// SIMATIC S7-200 project (STEP 7-Micro/WIN), CPU 224XP CN REL 02.01

SYMBOL_TABLE USR1
CRC_value        VW2070   // CRC的计算值
CRC_value_out    VW2090   // 调用CRC计算子程序得出的CRC值
TIMES_SENT       VB2001   // 发送记数寄存器
BYTES_REC        VB2002   // 接收的字节数
DATA_SENT        VB2010   // 发送区的起始字节
ADDRESS          VB2031   // 仪表地址
PORT_NUM         VB2005   // 选择的通信端口（PORT0 或PORT1）
END_SYMBOL_TABLE

SYMBOL_TABLE DI
紧急停止             I0.0
电源故障             I0.1
远程启动             I0.2
远程停止             I0.3
END_SYMBOL_TABLE

SYMBOL_TABLE USS 协议
USS_LOW_V        VD1000   // (DWORD)在此键入 USS协议符号的起始地址。
USS_HIGH_V       VD1004
USS_TIME_OUT     VW1008
USS_I_LINE       VW1010
USS_DAT_PTR0     VD1012
USS_ACT_DRV0     VD1016
USS_CUR_DRV0     VD1020
USS_P0           V1024.0
USS_REQ_SNT0     V1024.1
USS_RETRY_P0     VB1025
USS_ERR_CODE     VB1026
USS_CS_D0        VD1027
USS_CS_W0        VW1027
USS_CS_W2        VW1029
USS_CS_B0        VB1027
USS_CS_B1        VB1028
USS_POLL_BUF     VB1031
USS_XMT_0        VB1046
USS_XMT_ADR0     VB1049
USS_X_STWD       VD1056
USS_X_BCC        VB1060
USS_X_DW1        VD1047
USS_X_DW5        VD1051
USS_X_DW9        VD1055
USS_X_DB13       VB1059
USS_RCV_BUF0     VB1061
USS_R_STX        VB1062
USS_R_LGE        VB1063
USS_R_ADR        VB1064
USS_R_STWD       VD1071
USS_R_DW1        VD1062
USS_R_DW5        VD1066
USS_R_DW9        VD1070
USS_R_W13        VW1074
USS_STAT_TAB     VB1076
USS_ADR_P0       VB1396
END_SYMBOL_TABLE

SYMBOL_TABLE DO
启动排架             Q0.0
启动空调             Q0.1
启动空压机            Q0.2
DF1Q             Q0.3
DF2Q             Q0.4
DF3Q             Q0.5
DF4Q             Q0.6
DF5Q             Q0.7
运行Q              Q1.0
报警Q              Q1.1
END_SYMBOL_TABLE

SYMBOL_TABLE  内部
清洗间隔时间           VW4      // 0-999.9s
自动清洗延迟时间         VW6      // 0-1440min
清洗次数             VW8
报警温度设置值          VW12
报警光强度设置值         VW14
报警液位设置值          VW16
电流高报警设定值         VW18
电压高报警设定值         VW20
电压低报警设定值         VW22
温度高停止运行设置值       VW26
温度降允许运行设置值       VW28
光强低_自动清洗设置值      VW30
液位低停止运行设置值       VW34
液位升允许运行设置值       VW36
状态字1_1           VW38
状态字1_2           VW40
状态字2_1           VW42
状态字2_2           VW44
状态字3_1           VW46
状态字3_2           VW48
状态字4_1           VW50
状态字4_2           VW52
其它报警字1           VW54
其它报警字2           VW56
其它报警字3           VW58
累计运行时间（秒）        VW66     // 0-60
累计运行时间（分）        VW68     // 0-60
累计运行时间（时）        VW70     // 0-32767
累计启动次数           VW72     // 0-32767
温度1实时值           VW74
温度2实时值           VW76
光强实时值            VW78
液位实时值            VW80
电压实时值            VW82
电流实时值            VW84
清洗用临时积存1         VW140
清洗用临时积存2         VW142
清洗用临时积存3已清洗次     VW144
模块1通信监测临时        VB150
模块2通信监测临时        VB151
模块3通信监测临时        VB152
模块4通信监测临时        VB153
模块5通信监测临时        VB154
模块6通信监测临时        VB155
温度控制允许           M2.0     // 0为禁止,1为允许
光强度控制允许          M2.1     // 0为禁止,1为允许
液位控制允许           M2.2     // 0为禁止,1为允许
系统控制模式           M2.3     // 0为本地,1为远程
清洗控制模式           M2.4     // 0为手动,1为自动
温度1异常高           M6.0
温度2异常高           M6.1
光强异常低            M6.2
液位异常低            M6.3
未设定清洗参数          M6.4
未设定灯管开参数         M6.5
未设定报警参数          M6.6
允许清洗             M7.0
允许启动灯管           M7.1
中断清洗运行           M7.2
中断灯管运行           M7.3
模块1通信故障          M8.0
模块2通信故障          M8.1
模块3通信故障          M8.2
模块4通信故障          M8.3
模块5通信故障          M8.4
模块6通信故障          M8.5
排架1镇流器故障         M8.6
排架2镇流器故障         M8.7
排架3镇流器故障         M9.0
排架4镇流器故障         M9.1
排架5镇流器故障         M9.2
排架6镇流器故障         M9.3
排架7镇流器故障         M9.4
排架8镇流器故障         M9.5
排架9镇流器故障         M9.6
排架10镇流器故障        M9.7
灯管启动中            M10.0
清洗中              M10.1
空调运行中            M10.2
空压机运行中           M10.3
灯管本地启动           M10.4
灯管本地停止           M10.5
灯管远程启动           M10.6
灯管远程停止           M10.7
开始清洗             M11.1
停止清洗             M11.2
空调启动             M11.3
空调停止             M11.4
报警复位             M11.5
总报警位             M12.0
温度1高报警           M12.1
温度2高报警           M12.2
光强低报警            M12.3
液位低报警            M12.4
I高报警             M12.5
U高报警             M12.6
U低报警             M12.7
电源故障报警           M13.0
温度1输入故障          M13.1
温度2输入故障          M13.2
光强输入故障           M13.3
液位输入故障           M13.4
I输入故障            M13.5
U输入故障            M13.6
状态字1_1映象         MW14
状态字1_2映象         MW16
状态字2_1映象         MW18
状态字2_2映象         MW20
状态字3_1映象         MW22
状态字3_2映象         MW24
状态字4_1映象         MW26
状态字4_2映象         MW28
END_SYMBOL_TABLE

SYMBOL_TABLE AI
温度1AIW           AIW0     // 4------20ma
光强AIW            AIW2     // 0------5v
温度2AIW           AIW4     // 4------20ma
水位AIW            AIW6     // 4------20ma
电压AIW            AIW8     // 4------20ma
电流AIW            AIW10    // 4------20ma
END_SYMBOL_TABLE

ORGANIZATION_BLOCK MAIN:OB1
TITLE= 西门子PLC   RS485通信控制程序 
// 2007-4-25      Ver1.0      by huangyz0810@163.com
// 2007-4-26      Ver1.1      by huangyz0810@163.com
// 2007-4-30      Ver1.2      by huangyz0810@163.com
// 2007-5-07      Ver1.3      by huangyz0810@163.com
// *************************************************************************************************************************************************
// 注：主程序包括以下程序调用：通信初始化（INIT）、仪表数据处理（DI_DATA）、控制程序（CONTROL）
//         一般设备的控制程序请写入到CONTROL子程序里面。
// 
//         VB2060----VB2099范围内的40个字节空间已经分配给CRC校验子程序,切勿在其它程序中占用,否则引起麻烦
// 
//         VB2000----VB2049范围内的60个字节空间已经分配给通信中断,指针,字节计数等程序,切勿在其它程序中占用,
//                        其中,VB2010----2029 为发送缓冲区
//                                 VB2030----2059 为接收缓冲区
// 
//          VB2100----VB2199范围内的100个字节空间已经分配给数据读取队列,切勿在其它程序中占用,
//                        其中,VB2100----2109 为第数据队列的中间缓冲区
//                                 VB2110----2119 为第一个数据队列
//                                 VB2120----2129 为第二个数据队列
//                                  其它类推。该范围内最多支持9个队列，即最多支持不超过9次通信的设备数量。
//                                 如果需要超过9次通信，需要在 VB2200或其它未使用区域再分配通信队列寄存区
// *************************************************************************************************************************************************
// 
BEGIN
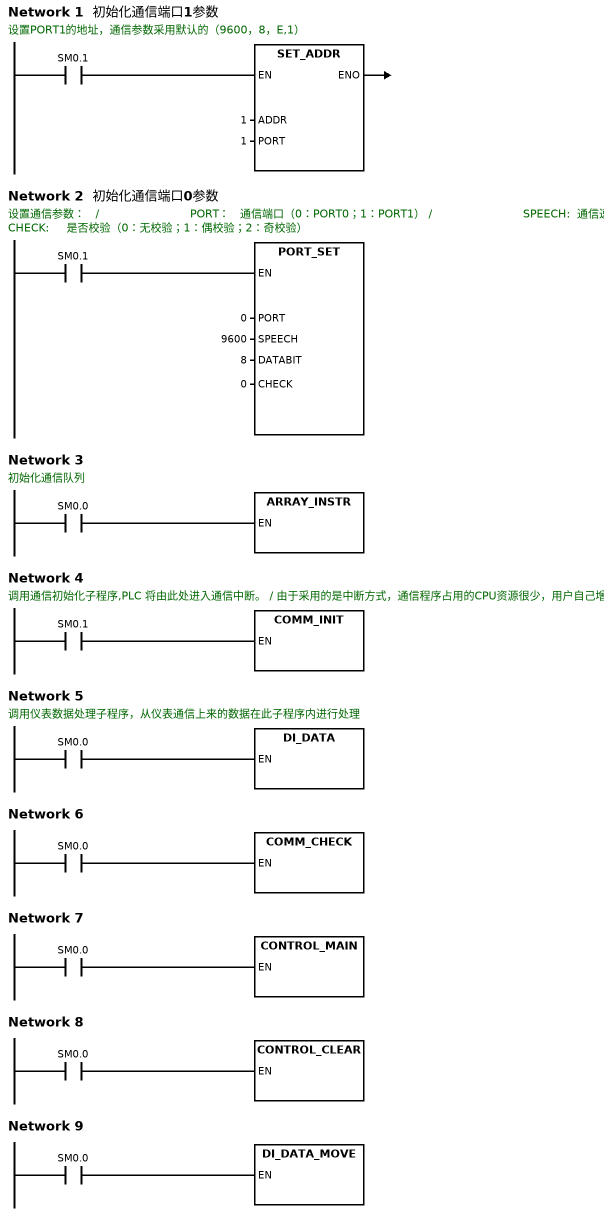
Network 1 // 初始化通信端口1参数
// 设置PORT1的地址，通信参数采用默认的（9600，8，E,1）
LD     SM0.1
SPA    1, 1
Network 2 // 初始化通信端口0参数
// 设置通信参数：  
//                          PORT：   通信端口（0：PORT0；1：PORT1）
//                          SPEECH:  通信速率（1200，2400，4800，9600，19200）
//                          DATABIT  :数据位（7或8）
//                          CHECK:     是否校验（0：无校验；1：偶校验；2：奇校验）
LD     SM0.1
CALL   PORT_SET:SBR55, 0, 9600, 8, 0
Network 3
// 初始化通信队列
LD     SM0.0
CALL   ARRAY_INSTR:SBR60
Network 4
// 调用通信初始化子程序,PLC 将由此处进入通信中断。
// 由于采用的是中断方式，通信程序占用的CPU资源很少，用户自己增加的程序可以很好的使用CPU资源
LD     SM0.1
CALL   COMM_INIT:SBR50
Network 5
// 调用仪表数据处理子程序，从仪表通信上来的数据在此子程序内进行处理
LD     SM0.0
CALL   DI_DATA:SBR52
Network 6
LD     SM0.0
CALL   COMM_CHECK:SBR53
Network 7
LD     SM0.0
CALL   CONTROL_MAIN:SBR1
Network 8
LD     SM0.0
CALL   CONTROL_CLEAR:SBR2
Network 9
LD     SM0.0
CALL   DI_DATA_MOVE:SBR6
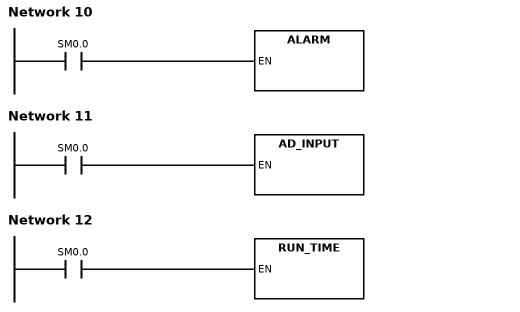
Network 10
LD     SM0.0
CALL   ALARM:SBR7
Network 11
LD     SM0.0
CALL   AD_INPUT:SBR8
Network 12
LD     SM0.0
CALL   RUN_TIME:SBR5
END_ORGANIZATION_BLOCK

SUBROUTINE_BLOCK CONTROL_MAIN:SBR1
TITLE=
BEGIN
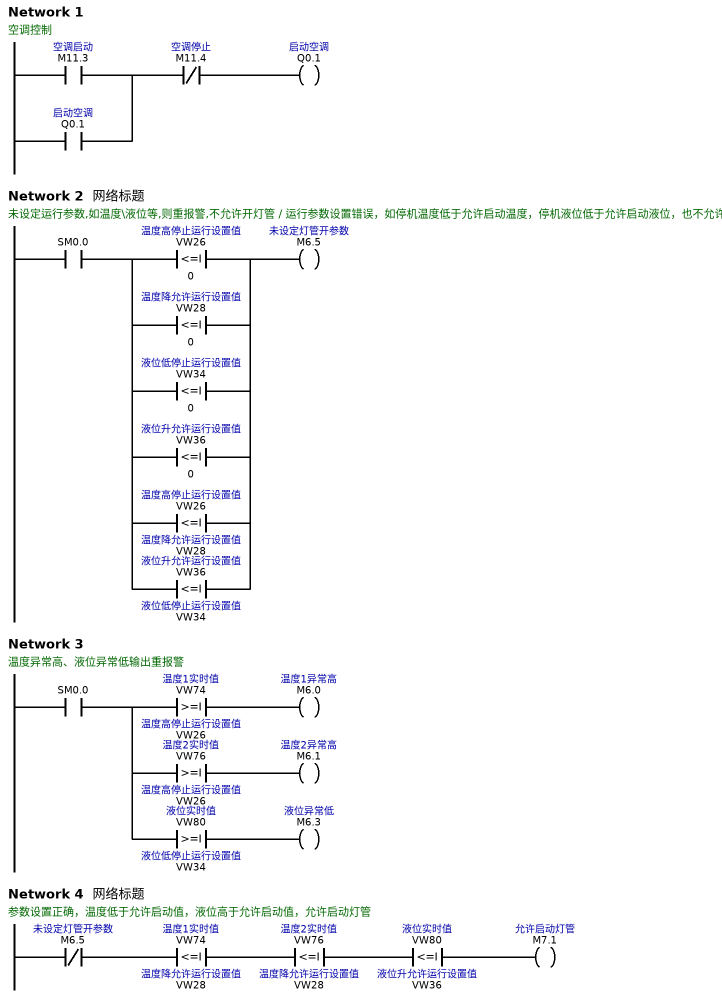
Network 1
// 空调控制
LD     空调启动:M11.3
O      启动空调:Q0.1
AN     空调停止:M11.4
=      启动空调:Q0.1
Network 2 // 网络标题
// 未设定运行参数,如温度\液位等,则重报警,不允许开灯管
// 运行参数设置错误，如停机温度低于允许启动温度，停机液位低于允许启动液位，也不允许开灯管
LD     SM0.0
LDW<=  温度高停止运行设置值:VW26, 0
OW<=   温度降允许运行设置值:VW28, 0
OW<=   液位低停止运行设置值:VW34, 0
OW<=   液位升允许运行设置值:VW36, 0
OW<=   温度高停止运行设置值:VW26, 温度降允许运行设置值:VW28
OW<=   液位升允许运行设置值:VW36, 液位低停止运行设置值:VW34
ALD
=      未设定灯管开参数:M6.5
Network 3
// 温度异常高、液位异常低输出重报警
LD     SM0.0
LPS
AW>=   温度1实时值:VW74, 温度高停止运行设置值:VW26
=      温度1异常高:M6.0
LRD
AW>=   温度2实时值:VW76, 温度高停止运行设置值:VW26
=      温度2异常高:M6.1
LPP
AW>=   液位实时值:VW80, 液位低停止运行设置值:VW34
=      液位异常低:M6.3
Network 4 // 网络标题
// 参数设置正确，温度低于允许启动值，液位高于允许启动值，允许启动灯管
LDN    未设定灯管开参数:M6.5
AW<=   温度1实时值:VW74, 温度降允许运行设置值:VW28
AW<=   温度2实时值:VW76, 温度降允许运行设置值:VW28
AW<=   液位实时值:VW80, 液位升允许运行设置值:VW36
=      允许启动灯管:M7.1
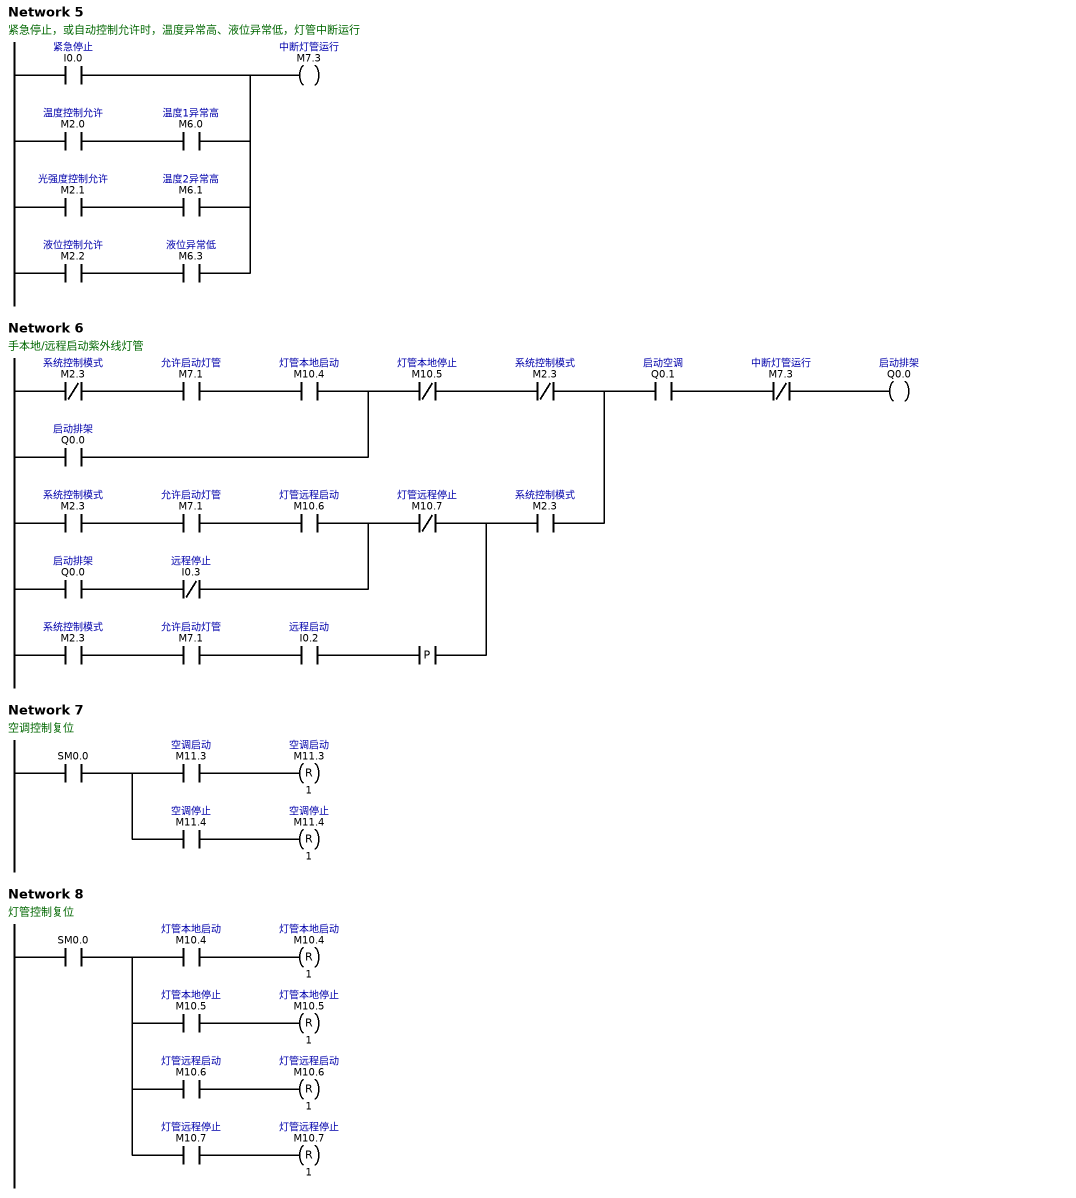
Network 5
// 紧急停止，或自动控制允许时，温度异常高、液位异常低，灯管中断运行
LD     紧急停止:I0.0
LD     温度控制允许:M2.0
A      温度1异常高:M6.0
OLD
LD     光强度控制允许:M2.1
A      温度2异常高:M6.1
OLD
LD     液位控制允许:M2.2
A      液位异常低:M6.3
OLD
=      中断灯管运行:M7.3
Network 6
// 手本地/远程启动紫外线灯管
LDN    系统控制模式:M2.3
A      允许启动灯管:M7.1
A      灯管本地启动:M10.4
O      启动排架:Q0.0
AN     灯管本地停止:M10.5
AN     系统控制模式:M2.3
LD     系统控制模式:M2.3
A      允许启动灯管:M7.1
A      灯管远程启动:M10.6
LD     启动排架:Q0.0
AN     远程停止:I0.3
OLD
AN     灯管远程停止:M10.7
LD     系统控制模式:M2.3
A      允许启动灯管:M7.1
A      远程启动:I0.2
EU
OLD
A      系统控制模式:M2.3
OLD
A      启动空调:Q0.1
AN     中断灯管运行:M7.3
=      启动排架:Q0.0
Network 7
// 空调控制复位
LD     SM0.0
LPS
A      空调启动:M11.3
R      空调启动:M11.3, 1
LPP
A      空调停止:M11.4
R      空调停止:M11.4, 1
Network 8
// 灯管控制复位
LD     SM0.0
LPS
A      灯管本地启动:M10.4
R      灯管本地启动:M10.4, 1
LRD
A      灯管本地停止:M10.5
R      灯管本地停止:M10.5, 1
LRD
A      灯管远程启动:M10.6
R      灯管远程启动:M10.6, 1
LPP
A      灯管远程停止:M10.7
R      灯管远程停止:M10.7, 1
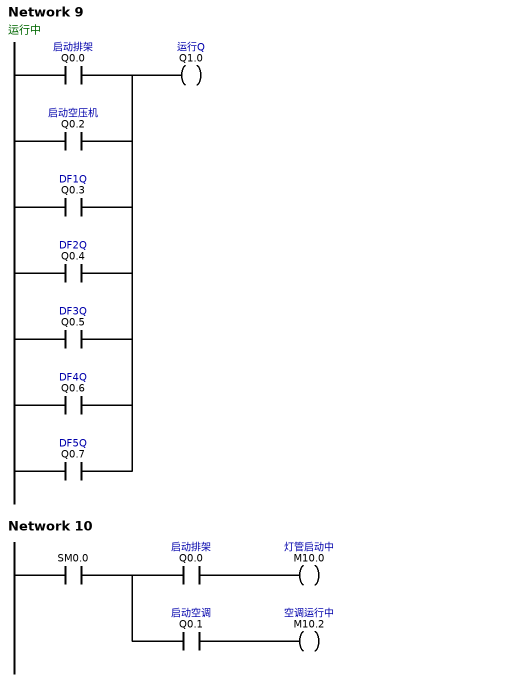
Network 9
// 运行中
LD     启动排架:Q0.0
O      启动空压机:Q0.2
O      DF1Q:Q0.3
O      DF2Q:Q0.4
O      DF3Q:Q0.5
O      DF4Q:Q0.6
O      DF5Q:Q0.7
=      运行Q:Q1.0
Network 10
LD     SM0.0
LPS
A      启动排架:Q0.0
=      灯管启动中:M10.0
LPP
A      启动空调:Q0.1
=      空调运行中:M10.2
END_SUBROUTINE_BLOCK

SUBROUTINE_BLOCK CONTROL_CLEAR:SBR2
TITLE=手动清洗, 清洗模式为"手动"后,先开空压机,延时5分钟,DF1输出10秒（值可调），停止10秒（值可调），反复3次，然后DF2输出10秒（值可调），停止10秒（值可调），反复3次，DF3、DF4、DF5照次类推
VAR
clean_time:WORD;	// LW0 
END_VAR
BEGIN
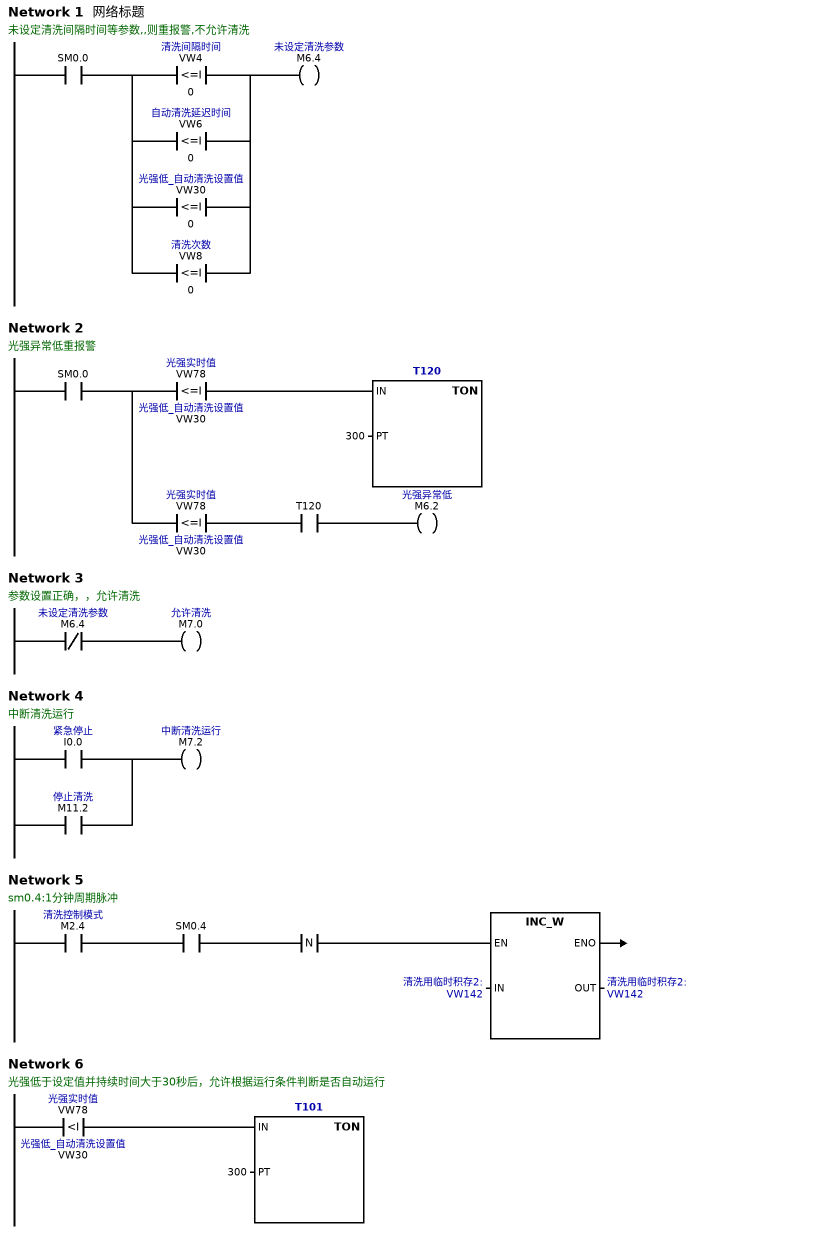
Network 1 // 网络标题
// 未设定清洗间隔时间等参数,,则重报警,不允许清洗
LD     SM0.0
LDW<=  清洗间隔时间:VW4, 0
OW<=   自动清洗延迟时间:VW6, 0
OW<=   光强低_自动清洗设置值:VW30, 0
OW<=   清洗次数:VW8, 0
ALD
=      未设定清洗参数:M6.4
Network 2
// 光强异常低重报警
LD     SM0.0
LPS
AW<=   光强实时值:VW78, 光强低_自动清洗设置值:VW30
TON    T120, 300
LPP
AW<=   光强实时值:VW78, 光强低_自动清洗设置值:VW30
A      T120
=      光强异常低:M6.2
Network 3
// 参数设置正确，，允许清洗
LDN    未设定清洗参数:M6.4
=      允许清洗:M7.0
Network 4
// 中断清洗运行
LD     紧急停止:I0.0
O      停止清洗:M11.2
=      中断清洗运行:M7.2
Network 5
// sm0.4:1分钟周期脉冲
LD     清洗控制模式:M2.4
A      SM0.4
ED
INCW   清洗用临时积存2:VW142
Network 6
// 光强低于设定值并持续时间大于30秒后，允许根据运行条件判断是否自动运行
LDW<   光强实时值:VW78, 光强低_自动清洗设置值:VW30
TON    T101, 300
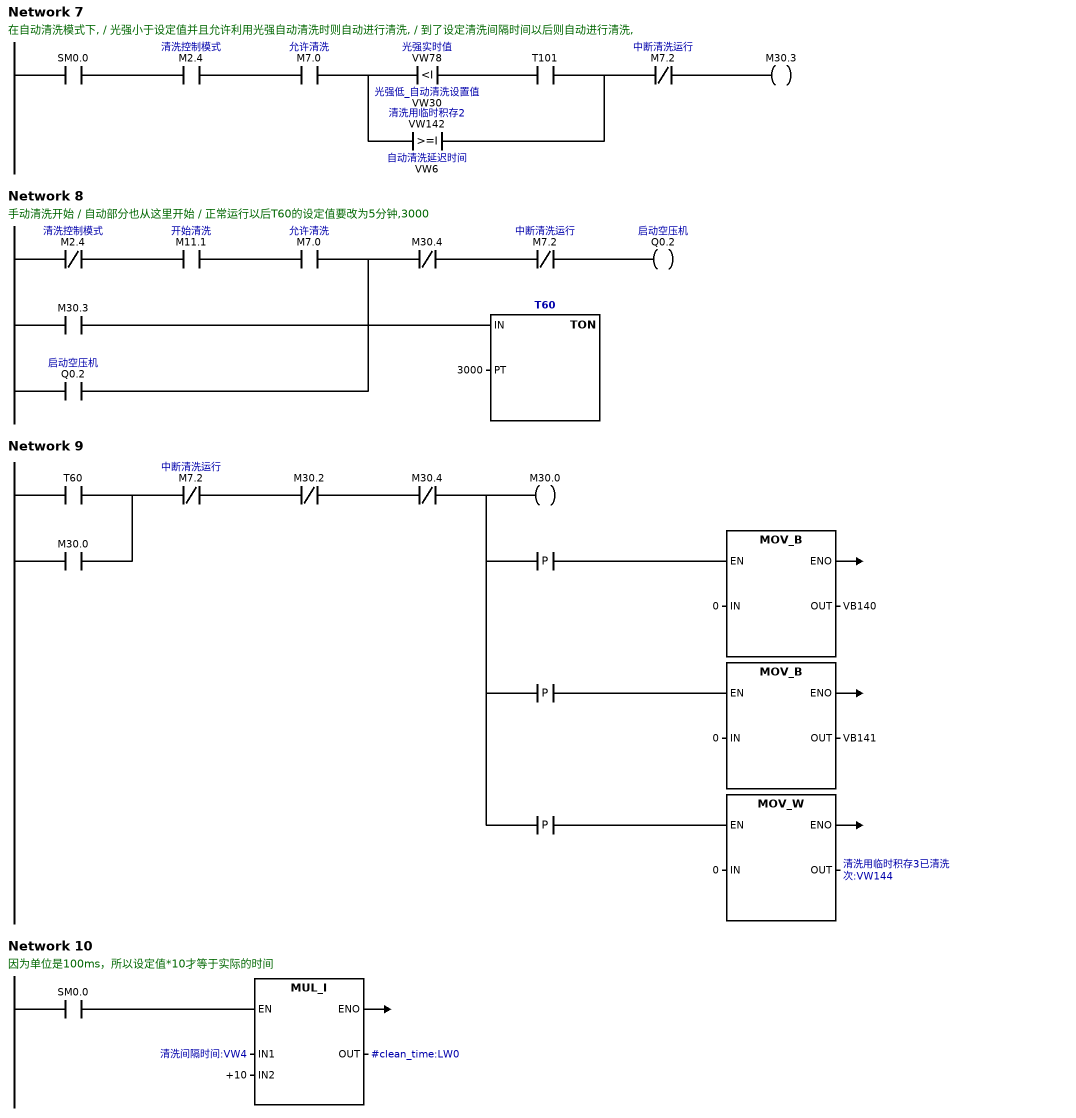
Network 7
// 在自动清洗模式下,
// 光强小于设定值并且允许利用光强自动清洗时则自动进行清洗,
// 到了设定清洗间隔时间以后则自动进行清洗,
LD     SM0.0
A      清洗控制模式:M2.4
A      允许清洗:M7.0
LDW<   光强实时值:VW78, 光强低_自动清洗设置值:VW30
A      T101
OW>=   清洗用临时积存2:VW142, 自动清洗延迟时间:VW6
ALD
AN     中断清洗运行:M7.2
=      M30.3
Network 8
// 手动清洗开始
// 自动部分也从这里开始
// 正常运行以后T60的设定值要改为5分钟,3000
LDN    清洗控制模式:M2.4
A      开始清洗:M11.1
A      允许清洗:M7.0
O      M30.3
O      启动空压机:Q0.2
LPS
AN     M30.4
AN     中断清洗运行:M7.2
=      启动空压机:Q0.2
LPP
TON    T60, 3000
Network 9
LD     T60
O      M30.0
AN     中断清洗运行:M7.2
AN     M30.2
AN     M30.4
LPS
=      M30.0
EU
MOVB   0, VB140
LRD
EU
MOVB   0, VB141
LPP
EU
MOVW   0, 清洗用临时积存3已清洗次:VW144
Network 10
// 因为单位是100ms，所以设定值*10才等于实际的时间
LD     SM0.0
MOVW   清洗间隔时间:VW4, #clean_time:LW0
*I     +10, #clean_time:LW0
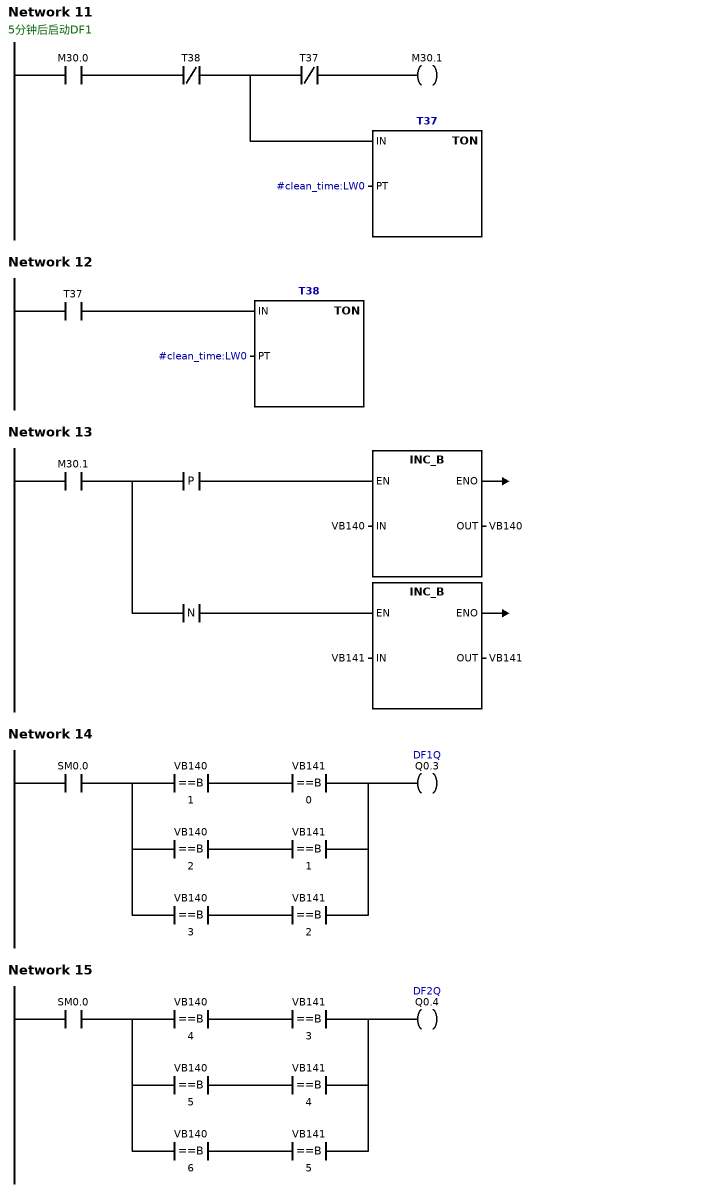
Network 11
// 5分钟后启动DF1
LD     M30.0
AN     T38
LPS
AN     T37
=      M30.1
LPP
TON    T37, #clean_time:LW0
Network 12
LD     T37
TON    T38, #clean_time:LW0
Network 13
LD     M30.1
LPS
EU
INCB   VB140
LPP
ED
INCB   VB141
Network 14
LD     SM0.0
LDB=   VB140, 1
AB=    VB141, 0
LDB=   VB140, 2
AB=    VB141, 1
OLD
LDB=   VB140, 3
AB=    VB141, 2
OLD
ALD
=      DF1Q:Q0.3
Network 15
LD     SM0.0
LDB=   VB140, 4
AB=    VB141, 3
LDB=   VB140, 5
AB=    VB141, 4
OLD
LDB=   VB140, 6
AB=    VB141, 5
OLD
ALD
=      DF2Q:Q0.4
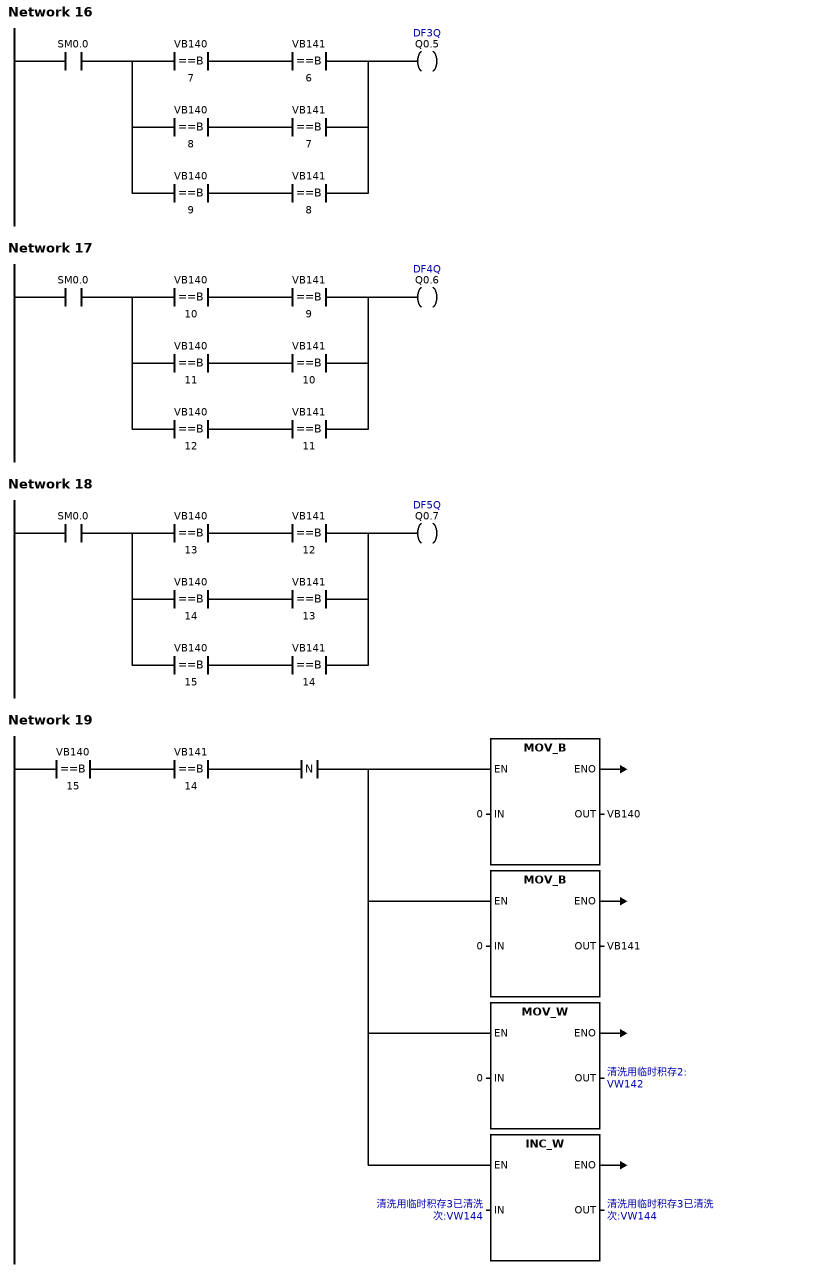
Network 16
LD     SM0.0
LDB=   VB140, 7
AB=    VB141, 6
LDB=   VB140, 8
AB=    VB141, 7
OLD
LDB=   VB140, 9
AB=    VB141, 8
OLD
ALD
=      DF3Q:Q0.5
Network 17
LD     SM0.0
LDB=   VB140, 10
AB=    VB141, 9
LDB=   VB140, 11
AB=    VB141, 10
OLD
LDB=   VB140, 12
AB=    VB141, 11
OLD
ALD
=      DF4Q:Q0.6
Network 18
LD     SM0.0
LDB=   VB140, 13
AB=    VB141, 12
LDB=   VB140, 14
AB=    VB141, 13
OLD
LDB=   VB140, 15
AB=    VB141, 14
OLD
ALD
=      DF5Q:Q0.7
Network 19
LDB=   VB140, 15
AB=    VB141, 14
ED
MOVB   0, VB140
MOVB   0, VB141
MOVW   0, 清洗用临时积存2:VW142
INCW   清洗用临时积存3已清洗次:VW144
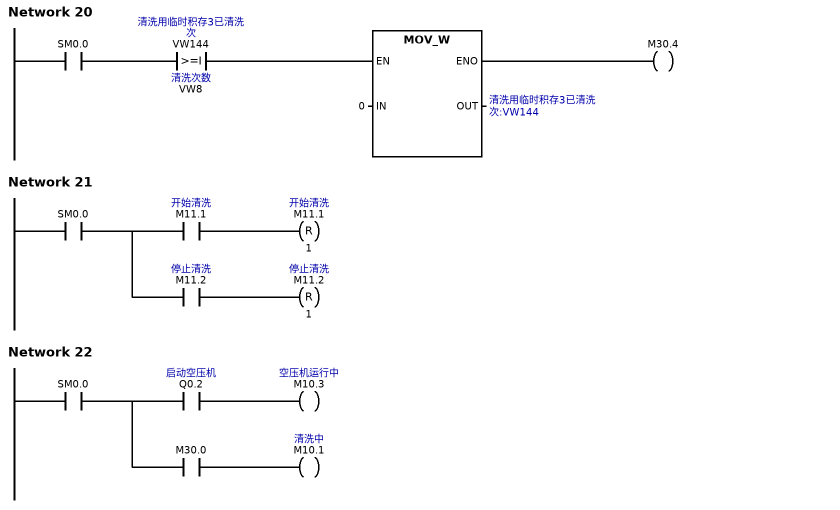
Network 20
LD     SM0.0
AW>=   清洗用临时积存3已清洗次:VW144, 清洗次数:VW8
MOVW   0, 清洗用临时积存3已清洗次:VW144
AENO
=      M30.4
Network 21
LD     SM0.0
LPS
A      开始清洗:M11.1
R      开始清洗:M11.1, 1
LPP
A      停止清洗:M11.2
R      停止清洗:M11.2, 1
Network 22
LD     SM0.0
LPS
A      启动空压机:Q0.2
=      空压机运行中:M10.3
LPP
A      M30.0
=      清洗中:M10.1
END_SUBROUTINE_BLOCK

SUBROUTINE_BLOCK RUN_TIME:SBR5
TITLE=系统运行后,每60秒暂时寄存器VW100自增1,每次计数达到60分,也就是1小时,运行总时间寄存器VW102自增1,VW100清零,重新计数.
BEGIN
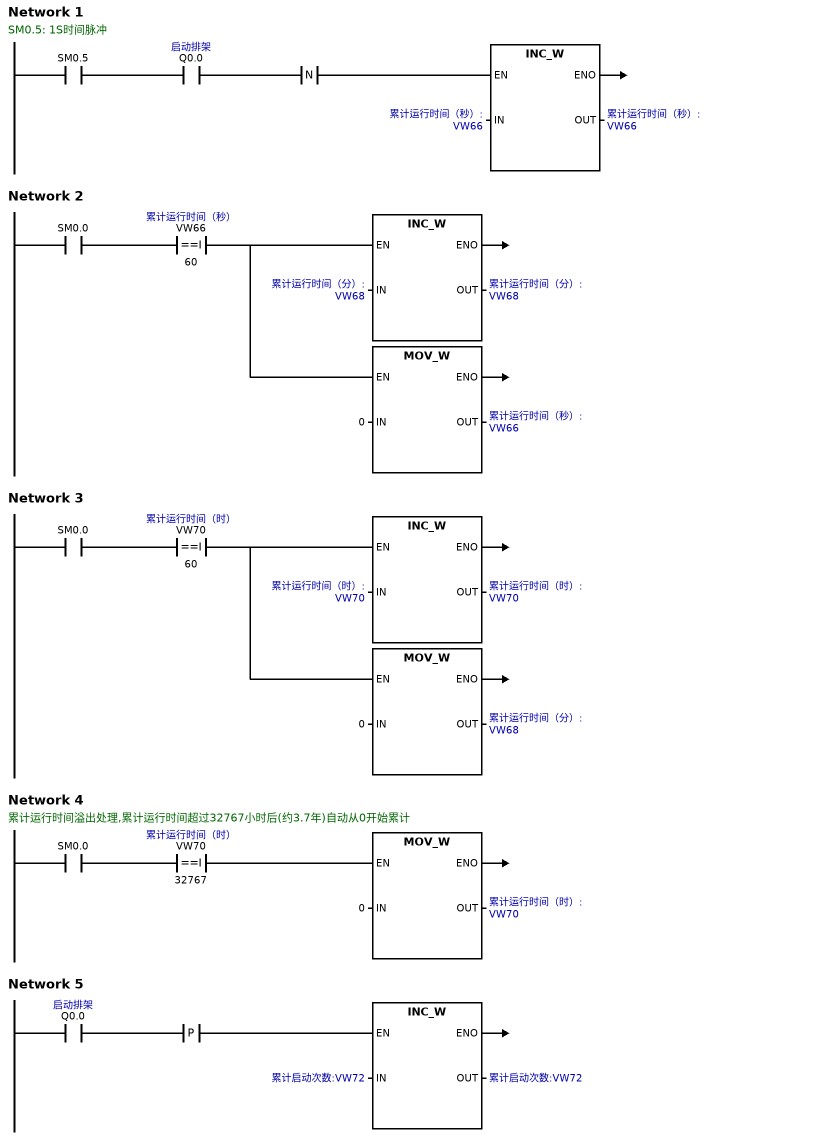
Network 1
// SM0.5: 1S时间脉冲
LD     SM0.5
A      启动排架:Q0.0
ED
INCW   累计运行时间（秒）:VW66
Network 2
LD     SM0.0
AW=    累计运行时间（秒）:VW66, 60
INCW   累计运行时间（分）:VW68
MOVW   0, 累计运行时间（秒）:VW66
Network 3
LD     SM0.0
AW=    累计运行时间（时）:VW70, 60
INCW   累计运行时间（时）:VW70
MOVW   0, 累计运行时间（分）:VW68
Network 4
// 累计运行时间溢出处理,累计运行时间超过32767小时后(约3.7年)自动从0开始累计
LD     SM0.0
AW=    累计运行时间（时）:VW70, 32767
MOVW   0, 累计运行时间（时）:VW70
Network 5
LD     启动排架:Q0.0
EU
INCW   累计启动次数:VW72
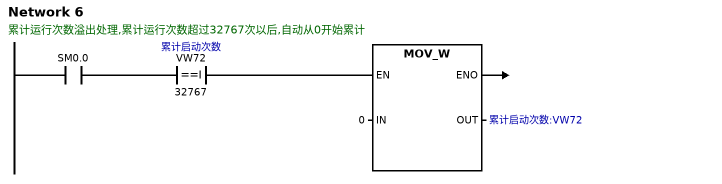
Network 6
// 累计运行次数溢出处理,累计运行次数超过32767次以后,自动从0开始累计
LD     SM0.0
AW=    累计启动次数:VW72, 32767
MOVW   0, 累计启动次数:VW72
Network 7 // 网络标题
// 网络注释
END_SUBROUTINE_BLOCK

SUBROUTINE_BLOCK DI_DATA_MOVE:SBR6
TITLE=子程序注释
BEGIN
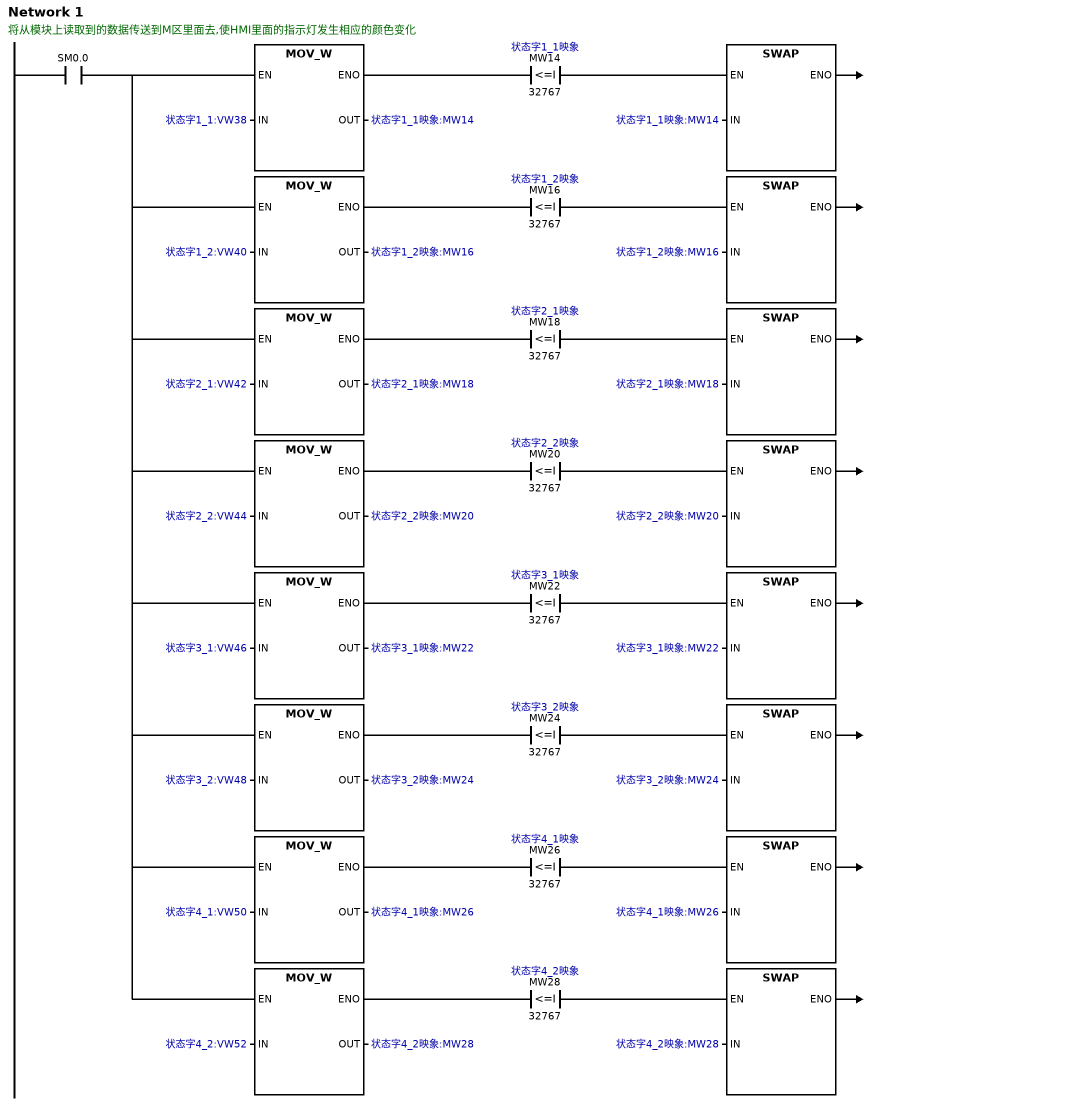
Network 1
// 将从模块上读取到的数据传送到M区里面去,使HMI里面的指示灯发生相应的颜色变化
LD     SM0.0
LPS
MOVW   状态字1_1:VW38, 状态字1_1映象:MW14
AENO
AW<=   状态字1_1映象:MW14, 32767
SWAP   状态字1_1映象:MW14
LRD
MOVW   状态字1_2:VW40, 状态字1_2映象:MW16
AENO
AW<=   状态字1_2映象:MW16, 32767
SWAP   状态字1_2映象:MW16
LRD
MOVW   状态字2_1:VW42, 状态字2_1映象:MW18
AENO
AW<=   状态字2_1映象:MW18, 32767
SWAP   状态字2_1映象:MW18
LRD
MOVW   状态字2_2:VW44, 状态字2_2映象:MW20
AENO
AW<=   状态字2_2映象:MW20, 32767
SWAP   状态字2_2映象:MW20
LRD
MOVW   状态字3_1:VW46, 状态字3_1映象:MW22
AENO
AW<=   状态字3_1映象:MW22, 32767
SWAP   状态字3_1映象:MW22
LRD
MOVW   状态字3_2:VW48, 状态字3_2映象:MW24
AENO
AW<=   状态字3_2映象:MW24, 32767
SWAP   状态字3_2映象:MW24
LRD
MOVW   状态字4_1:VW50, 状态字4_1映象:MW26
AENO
AW<=   状态字4_1映象:MW26, 32767
SWAP   状态字4_1映象:MW26
LPP
MOVW   状态字4_2:VW52, 状态字4_2映象:MW28
AENO
AW<=   状态字4_2映象:MW28, 32767
SWAP   状态字4_2映象:MW28
END_SUBROUTINE_BLOCK

SUBROUTINE_BLOCK ALARM:SBR7
TITLE=报警
VAR
alarm_temp1:BOOL;	// L0.0 
alarm_temp2:BOOL;	// L0.1 
alarm_temp3:BOOL;	// L0.2 
END_VAR
BEGIN
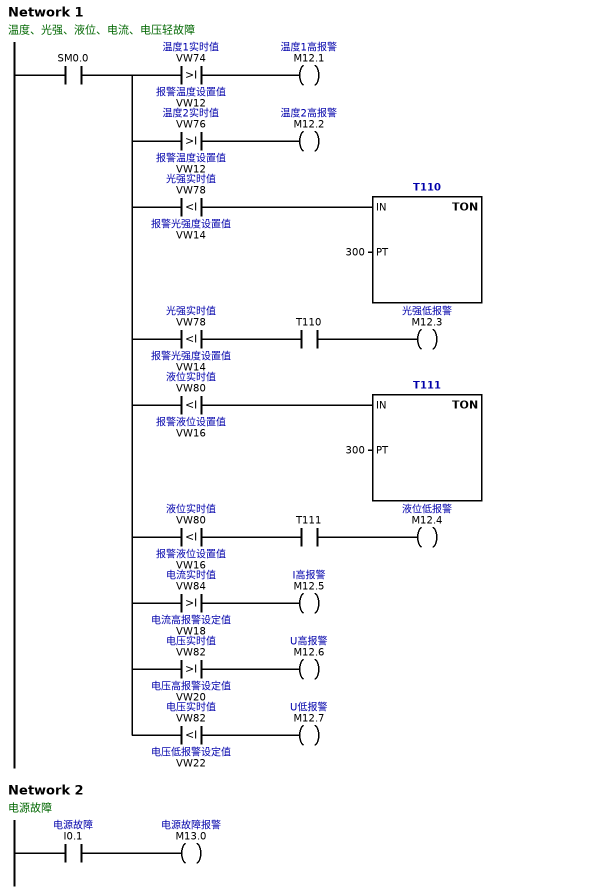
Network 1
// 温度、光强、液位、电流、电压轻故障
LD     SM0.0
LPS
AW>    温度1实时值:VW74, 报警温度设置值:VW12
=      温度1高报警:M12.1
LRD
AW>    温度2实时值:VW76, 报警温度设置值:VW12
=      温度2高报警:M12.2
LRD
AW<    光强实时值:VW78, 报警光强度设置值:VW14
TON    T110, 300
LRD
AW<    光强实时值:VW78, 报警光强度设置值:VW14
A      T110
=      光强低报警:M12.3
LRD
AW<    液位实时值:VW80, 报警液位设置值:VW16
TON    T111, 300
LRD
AW<    液位实时值:VW80, 报警液位设置值:VW16
A      T111
=      液位低报警:M12.4
LRD
AW>    电流实时值:VW84, 电流高报警设定值:VW18
=      I高报警:M12.5
LRD
AW>    电压实时值:VW82, 电压高报警设定值:VW20
=      U高报警:M12.6
LPP
AW<    电压实时值:VW82, 电压低报警设定值:VW22
=      U低报警:M12.7
Network 2
// 电源故障
LD     电源故障:I0.1
=      电源故障报警:M13.0
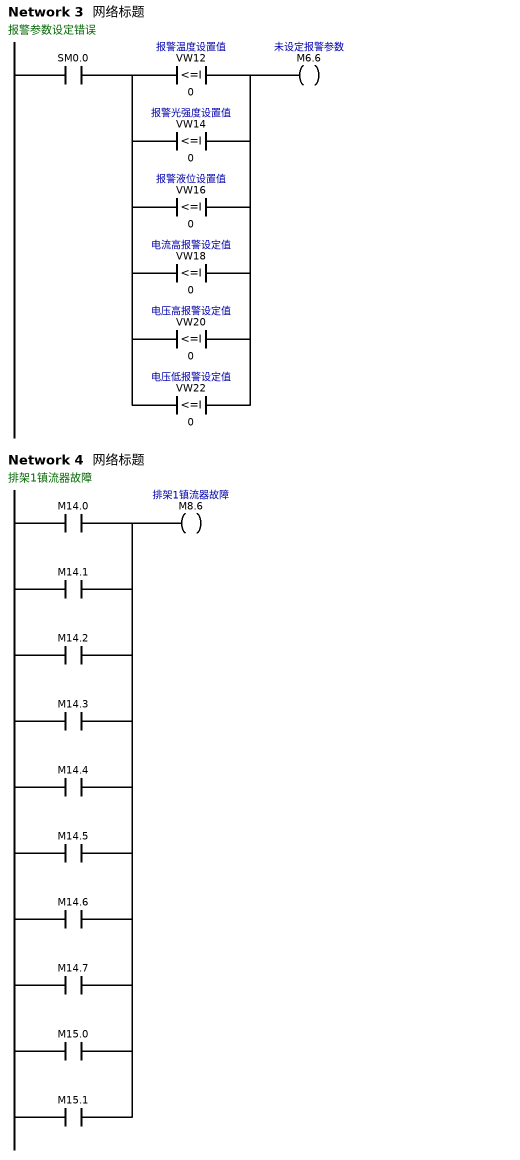
Network 3 // 网络标题
// 报警参数设定错误
LD     SM0.0
LDW<=  报警温度设置值:VW12, 0
OW<=   报警光强度设置值:VW14, 0
OW<=   报警液位设置值:VW16, 0
OW<=   电流高报警设定值:VW18, 0
OW<=   电压高报警设定值:VW20, 0
OW<=   电压低报警设定值:VW22, 0
ALD
=      未设定报警参数:M6.6
Network 4 // 网络标题
// 排架1镇流器故障
LD     M14.0
O      M14.1
O      M14.2
O      M14.3
O      M14.4
O      M14.5
O      M14.6
O      M14.7
O      M15.0
O      M15.1
=      排架1镇流器故障:M8.6
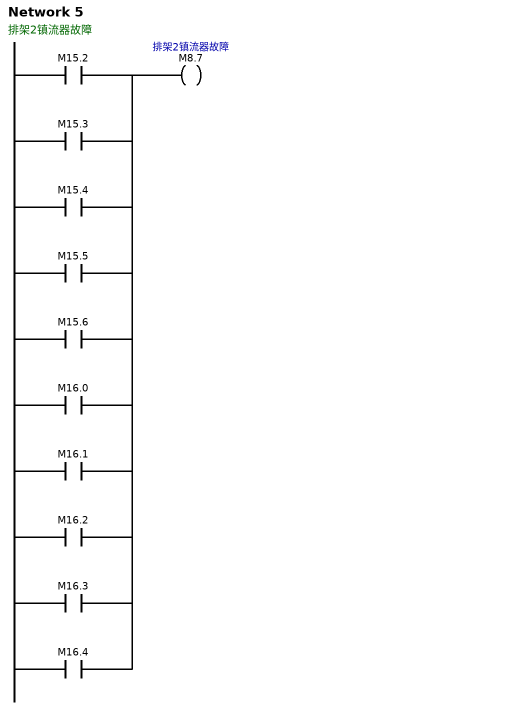
Network 5
// 排架2镇流器故障
LD     M15.2
O      M15.3
O      M15.4
O      M15.5
O      M15.6
O      M16.0
O      M16.1
O      M16.2
O      M16.3
O      M16.4
=      排架2镇流器故障:M8.7
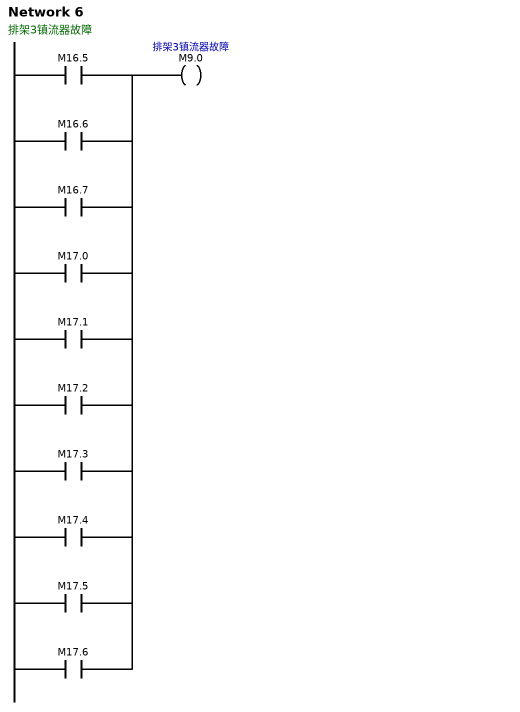
Network 6
// 排架3镇流器故障
LD     M16.5
O      M16.6
O      M16.7
O      M17.0
O      M17.1
O      M17.2
O      M17.3
O      M17.4
O      M17.5
O      M17.6
=      排架3镇流器故障:M9.0
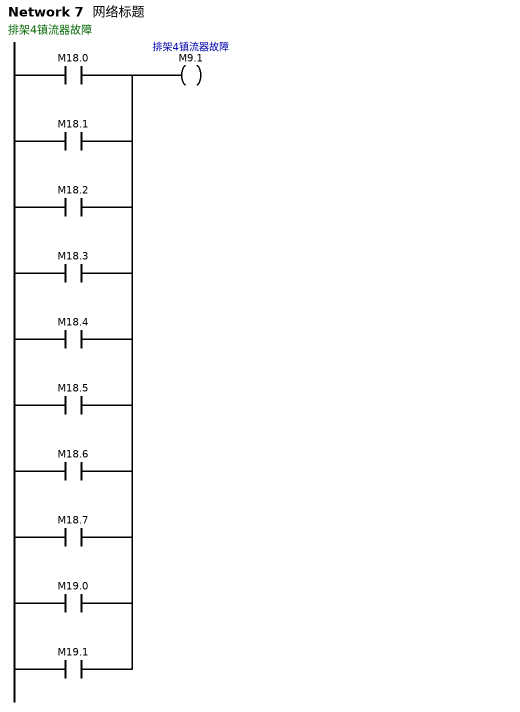
Network 7 // 网络标题
// 排架4镇流器故障
LD     M18.0
O      M18.1
O      M18.2
O      M18.3
O      M18.4
O      M18.5
O      M18.6
O      M18.7
O      M19.0
O      M19.1
=      排架4镇流器故障:M9.1
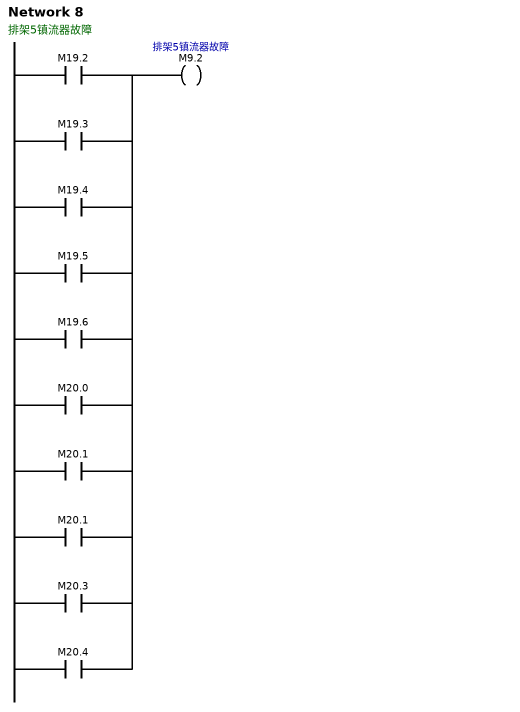
Network 8
// 排架5镇流器故障
LD     M19.2
O      M19.3
O      M19.4
O      M19.5
O      M19.6
O      M20.0
O      M20.1
O      M20.1
O      M20.3
O      M20.4
=      排架5镇流器故障:M9.2
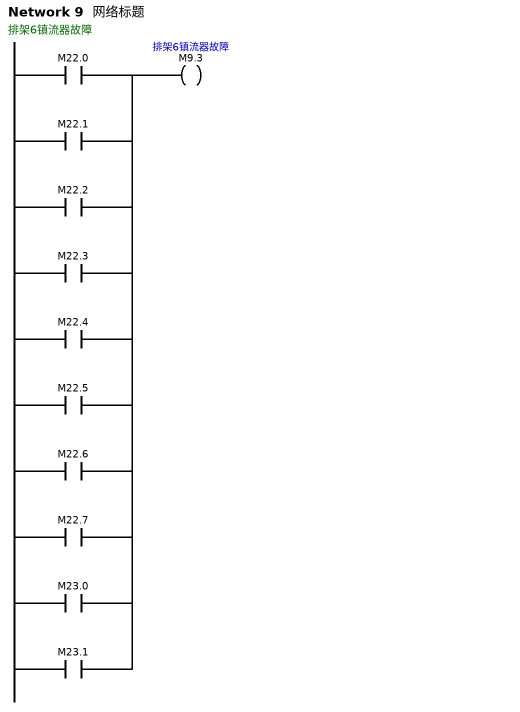
Network 9 // 网络标题
// 排架6镇流器故障
LD     M22.0
O      M22.1
O      M22.2
O      M22.3
O      M22.4
O      M22.5
O      M22.6
O      M22.7
O      M23.0
O      M23.1
=      排架6镇流器故障:M9.3
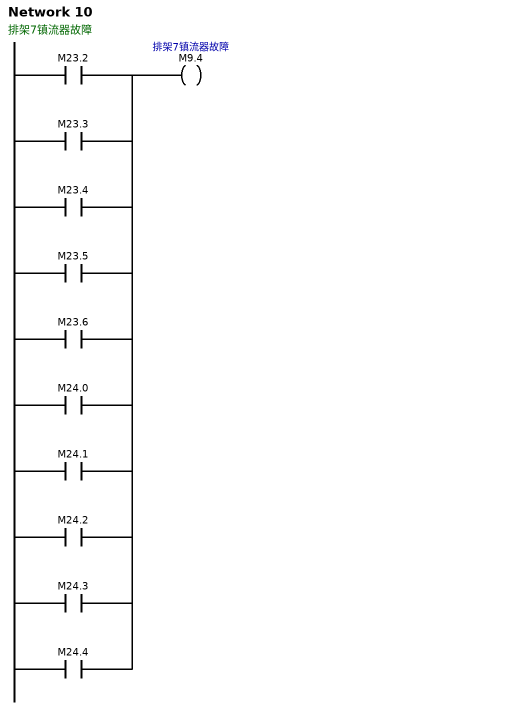
Network 10
// 排架7镇流器故障
LD     M23.2
O      M23.3
O      M23.4
O      M23.5
O      M23.6
O      M24.0
O      M24.1
O      M24.2
O      M24.3
O      M24.4
=      排架7镇流器故障:M9.4
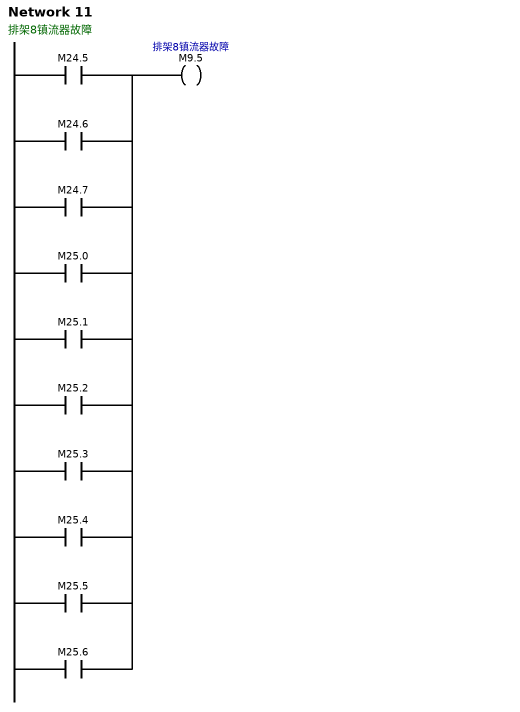
Network 11
// 排架8镇流器故障
LD     M24.5
O      M24.6
O      M24.7
O      M25.0
O      M25.1
O      M25.2
O      M25.3
O      M25.4
O      M25.5
O      M25.6
=      排架8镇流器故障:M9.5
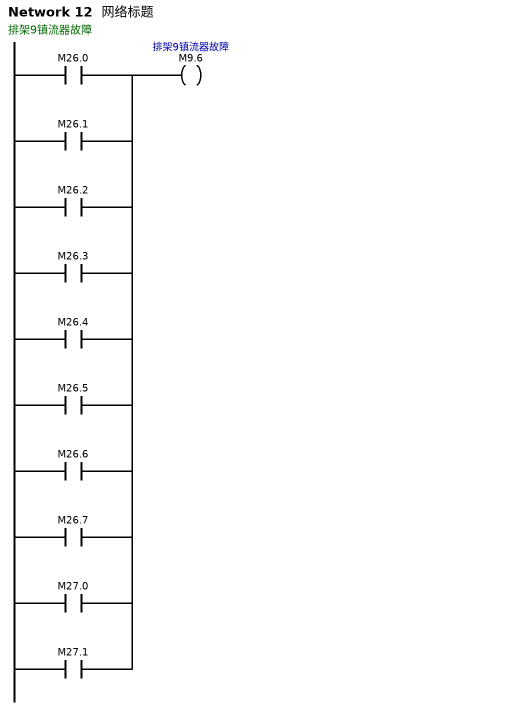
Network 12 // 网络标题
// 排架9镇流器故障
LD     M26.0
O      M26.1
O      M26.2
O      M26.3
O      M26.4
O      M26.5
O      M26.6
O      M26.7
O      M27.0
O      M27.1
=      排架9镇流器故障:M9.6
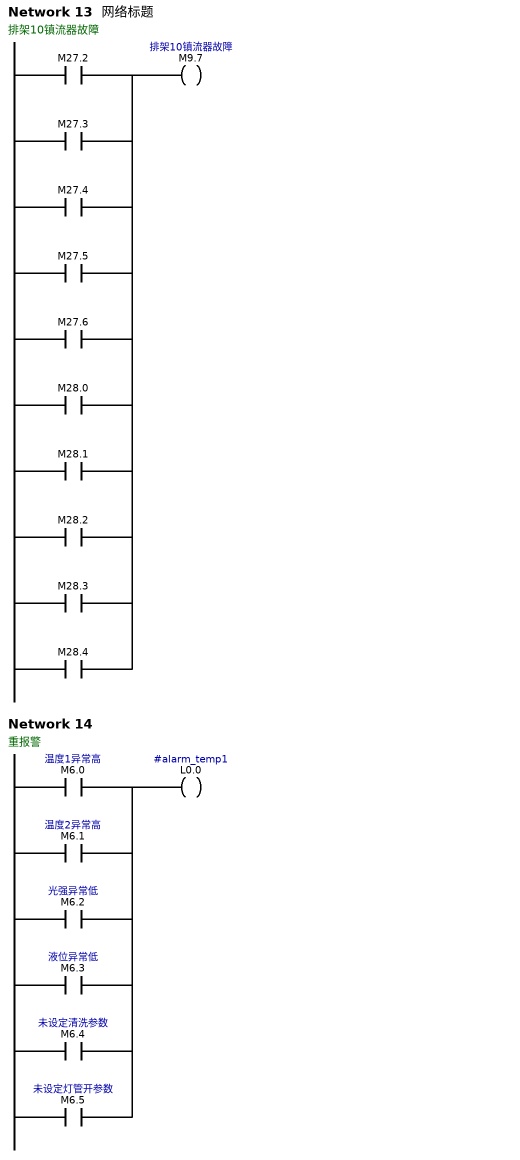
Network 13 // 网络标题
// 排架10镇流器故障
LD     M27.2
O      M27.3
O      M27.4
O      M27.5
O      M27.6
O      M28.0
O      M28.1
O      M28.2
O      M28.3
O      M28.4
=      排架10镇流器故障:M9.7
Network 14
// 重报警
LD     温度1异常高:M6.0
O      温度2异常高:M6.1
O      光强异常低:M6.2
O      液位异常低:M6.3
O      未设定清洗参数:M6.4
O      未设定灯管开参数:M6.5
=      #alarm_temp1:L0.0
